// TwinCAT 3 PLC project Untitled1
// Title: FileReadWriteOpen
// Company: Changdae
// Author: Back, Changdae
// ProjectVersion: 1.0
// Description: Simple File Read, Write, Open via HMI
// ProgramVersion: 3.1.4024.12
// libraries:
//   Tc2_Standard, * (Beckhoff Automation GmbH)
//   Tc2_System, * (Beckhoff Automation GmbH)
//   Tc2_Utilities, * (Beckhoff Automation GmbH)
//   Tc3_Module, * (Beckhoff Automation GmbH)
// project tree:
//   / PlcTask.TcTTO
//   POUs/ FB_FileGenerator.TcPOU, FB_FileReader.TcPOU, FB_OpenFileFromWindow.TcPOU, MAIN.TcPOU

CONFIGURATION Untitled1
    RESOURCE PLC ON TwinCAT3
        TASK PlcTask(INTERVAL := T#10ms, PRIORITY := 20);
        PROGRAM MAIN WITH PlcTask : MAIN;
    END_RESOURCE
END_CONFIGURATION

// ---- POUs/MAIN.TcPOU
PROGRAM MAIN
VAR
	fbFileGenerator 		: FB_FileGenerator;	
	fbFileReader 			: FB_FileReader;
	fbOpenFileFromWindow	: FB_OpenFileFromWindow;
	
	(* HMI Interface variable *)
	sFileName_HI	: STRING(70);
	sSelectedFile_HI : STRING(70);
	sSelectedDirectory_HI : STRING(170);	
END_VAR

fbFileGenerator(sSelectedDirectory := sSelectedDirectory_HI, sFileName := sFileName_HI);
fbFileReader(sSelectedFile := sSelectedFile_HI ,sSelectedDirectory := sSelectedDirectory_HI);
fbOpenFileFromWindow(sSelectedFile := sSelectedFile_HI, sSelectedDirectory := sSelectedDirectory_HI);

END_PROGRAM

// ---- POUs/FB_FileGenerator.TcPOU
FUNCTION_BLOCK FB_FileGenerator
VAR_INPUT
	sFileName : STRING(70);
	sSelectedDirectory : STRING(170);
	sSomethingToWrite : STRING(1024);
	bExecute : BOOL;
END_VAR

VAR_OUTPUT
	bError : BOOL;
	nErrorID : UDINT;
END_VAR

VAR
	fbFileOpen : FB_FileOpen :=(nMode := FOPEN_MODEWRITE, ePath := PATH_GENERIC);
	fbFileWrite : FB_FileWrite;
	fbFileClose : FB_FileClose;
	rTrigExecute : R_TRIG;
	sErrorState : STRING;
	eState : (Init, FileOpening, FileWriting, FileClosing, Error);
	
END_VAR

rTrigExecute(CLK:=bExecute);

CASE eState OF
	Init:
		fbFileOpen(bExecute := FALSE);	
	    fbFileWrite(bExecute := FALSE);
	    fbFileClose(bExecute := FALSE);
		nErrorID := 0;
		bError := FALSE;
		
		IF rTrigExecute.Q THEN
			eState := FileOpening;
		END_IF
	
	FileOpening:
		fbFileOpen(bExecute := TRUE,
					sPathName := CONCAT(GetDirectoryPath(sSelectedDirectory),sFileName));
		IF fbFileOpen.bError THEN
			nErrorID := fbFileOpen.nErrId;
			eState := Error;	
			sErrorState := 'FileOpening';
		ELSIF NOT fbFileOpen.bBusy THEN
			fbFileOpen(bExecute := FALSE);
			eState := FileWriting;
		END_IF
		
	FileWriting:
		fbFileWrite(bExecute := TRUE,
					hFile:= fbFileOpen.hFile,
					pWriteBuff:=ADR(sSomethingToWrite),
					cbWriteLen := SIZEOF(sSomethingToWrite));
		IF fbFileWrite.bError THEN
			eState := Error;
			nErrorID := fbFileWrite.nErrId;
			sErrorState := 'FileWriting';
		ELSIF NOT fbFileWrite.bBusy THEN
			fbFileWrite(bExecute := FALSE);
			eState := FileClosing;
		END_IF
	
	FileClosing:
		fbFileClose(bExecute := TRUE,
					hFile := fbFileOpen.hFile);
		IF fbFileClose.bError THEN
			nErrorID := fbFileClose.nErrId;
			eState := Error;
			sErrorState := 'FileClosing';	
		ELSIF NOT fbFileClose.bBusy THEN
			eState := Init;
		END_IF
	
	Error:
		bError := TRUE;
		IF rTrigExecute.Q THEN
			eState := Init;
		END_IF
END_CASE

METHOD PRIVATE GetDirectoryPath : STRING
VAR_INPUT
	sSelectedDirectroy : STRING(170);
END_VAR
VAR
	
END_VAR
VAR CONSTANT
	sCdrive : STRING(3) := 'C:\';
	sSlash : STRING(1) := '/';
END_VAR
GetDirectoryPath := CONCAT(sCdrive, sSelectedDirectroy);
GetDirectoryPath := CONCAT(GetDirectoryPath, sSlash);

(* Return: C:\xxx/ *)
END_METHOD

END_FUNCTION_BLOCK

// ---- POUs/FB_FileReader.TcPOU
FUNCTION_BLOCK FB_FileReader
VAR_INPUT
	sSelectedFile : STRING(70);
	sSelectedDirectory : STRING(170);
	bExecute : BOOL;
END_VAR
VAR_OUTPUT
	bError : BOOL;
	
	(*ADS Error Return code*)
	nErrorID : UDINT;
END_VAR
VAR
	fbFileOpen : FB_FileOpen := (nMode := FOPEN_MODEREAD, ePath := PATH_GENERIC);
	fbFileRead : FB_FileRead;
	fbFileClose : FB_FileClose;
	rTrigExecute : R_TRIG;
	eState : (Init, FileOpening, FileReading, FileClosing, Error);	
	sErrorState : STRING;
	
	sSomethingToRead : STRING(1024);
END_VAR

rTrigExecute(CLK:=bExecute);

CASE eState OF
	Init:
		fbFileOpen(bExecute := FALSE);
		fbFileRead(bExecute := FALSE);
		fbFileClose(bExecute := FALSE);
		bError := FALSE;
		nErrorID := 0;
		IF rTrigExecute.Q THEN
			eState:=FileOpening;
			sSomethingToRead := '';
		END_IF
		
	FileOpening:
		fbFileOpen(bExecute := TRUE,
					sPathName := CONCAT(GetDirectoryPath(sSelectedDirectory),GetFileName(sSelectedFile)));
		IF fbFileOpen.bError THEN
			nErrorID := fbFileOpen.nErrId;
			eState := Error;	
			sErrorState := 'FileOpening';
		ELSIF NOT fbFileOpen.bBusy THEN
			fbFileOpen(bExecute := FALSE);
			eState := FileReading;
		END_IF
		

	FileReading:
		fbFileRead(bExecute := TRUE,
					hFile := fbFileOpen.hFile,
					pReadBuff := ADR(sSomethingToRead),
					cbReadLEN := SIZEOF(sSomethingToRead) - 1);
		IF fbFileRead.bError THEN
			nErrorID := fbFileRead.nErrId;
			sErrorState := 'FileReading';
			eState := Error;	
		ELSIF NOT fbFileRead.bBusy THEN
			fbFileRead(bExecute := FALSE);
			eState := FileClosing;
		END_IF
	
	FileClosing:
		fbFileClose(bExecute := TRUE,
					hFile := fbFileOpen.hFile);
		IF fbFileClose.bError THEN
			nErrorID := fbFileClose.nErrId;
			eState := Error;
			sErrorState := 'FileClosing';	
		ELSIF NOT fbFileClose.bBusy THEN
			eState := Init;
		END_IF
	
	Error:
		bError := TRUE;
		IF rTrigExecute.Q THEN
			eState := Init;
		END_IF
END_CASE

METHOD PRIVATE GetDirectoryPath : STRING
VAR_INPUT
	sSelectedDirectroy : STRING(170);
END_VAR
VAR
	
END_VAR
VAR CONSTANT
	sCdrive : STRING(3) := 'C:\';
	sSlash : STRING(1) := '/';
END_VAR
GetDirectoryPath := CONCAT(sCdrive, sSelectedDirectroy);
GetDirectoryPath := CONCAT(GetDirectoryPath, sSlash);

(* Return: C:\xxx/ *)
END_METHOD

METHOD PRIVATE GetFileName : STRING
VAR_INPUT
	sSelectedFile : STRING(70);
END_VAR
GetFileName := DELETE(sSelectedFile,2,LEN(sSelectedFile)-1);
GetFileName := DELETE(GetFileName,2,1);
END_METHOD

END_FUNCTION_BLOCK

// ---- POUs/FB_OpenFileFromWindow.TcPOU
FUNCTION_BLOCK FB_OpenFileFromWindow
VAR_INPUT
	sSelectedFile : STRING(70);
	sSelectedDirectory : STRING(170);
	bExecute : BOOL;
END_VAR
VAR_OUTPUT
	bError : BOOL;
	nErrorID : UDINT;
END_VAR
VAR
	fbStartProcess : NT_StartProcess := (PATHSTR := 'C:\Windows\System32\notepad.exe' );
	rTrigExecute : R_trig;
	eState : (Init, StartNotePad, Error);
END_VAR

rTrigExecute(CLK:=bExecute);

CASE eState OF
	Init:
		fbStartProcess(START:=FALSE);
		bError := FALSE;
		nErrorID := 0;
		IF rTrigExecute.Q THEN
			eState := StartNotePad;
		END_IF
	
	StartNotePad:
		fbStartProcess(
						START := TRUE, 
						DIRNAME := GetDirectoryPath(sSelectedDirectroy := sSelectedDirectory),
						COMNDLINE := GetFileName(sSelectedFile := sSelectedFile)
						);
		IF fbStartProcess.ERR THEN
			eState := Error;
			bError := TRUE;
			nErrorID := fbStartProcess.ERRID;
		ELSIF NOT fbStartProcess.BUSY THEN
			eState := Init;
		END_IF
 
	Error:
		IF rTrigExecute.Q THEN
			eState := Init;
		END_IF	
END_CASE

METHOD PRIVATE GetDirectoryPath : STRING
VAR_INPUT
	sSelectedDirectroy : STRING(170);
END_VAR
VAR
	
END_VAR
VAR CONSTANT
	sCdrive : STRING(3) := 'C:\';
	sSlash : STRING(1) := '/';
END_VAR
GetDirectoryPath := CONCAT(sCdrive, sSelectedDirectroy);
GetDirectoryPath := CONCAT(GetDirectoryPath, sSlash);

(* Result : C:\sSelctedDirectory/ *)
END_METHOD

METHOD PRIVATE GetFileName : STRING
VAR_INPUT
	sSelectedFile : STRING(70);
END_VAR
GetFileName := DELETE(sSelectedFile,2,LEN(sSelectedFile)-1);
GetFileName := DELETE(GetFileName,2,1);
END_METHOD

END_FUNCTION_BLOCK
